FUNCTION_BLOCK L3_PlatoDivisor EXTENDS L1_ModuleBase

VAR_OUTPUT	
	fbController	: L2_PlatoDivisor_SFC:=(dr:=dr);  
	d0 				: L1_Sensor := (uiValue:= TRUE);
    D_1       		: L1_Actuator;
    E_1       		: L1_Actuator;
	NumGiros 		: DINT := 0;
	Angulo			: REAL := 0;
END_VAR

VAR
	AnguloAnim		: REAL := 0;
END_VAR

METHOD ProcessCycle : BOOL 

VAR_INPUT
	dr			: REFERENCE TO L1_Director;
	tapas		: REFERENCE TO L6_Tapas;	
END_VAR
IF dr.gmModeActual = L1_GEMMA.A6Inicializando THEN
	NumGiros := 0;
	Angulo	 := 0; // -45.0;
ELSE
	// Sensores y condiciones iniciales
	d0.ProcessCycle(LocalHost:=dr.gmLocalHost, sfcValue=>fbController.d0);
	IC := d0.uiValue;
	
	// Controlador
	fbController.ProcessCycle(dr.gmModeActual);
	fbController(
		dr:=dr, IC:=IC, Execute:=Execute, Ack:=Ack, Ready=>Ready, Done=>Done);
	IF fbController.Done AND NOT fbController.Performed THEN
		fbController.Performed 	:= TRUE;
		NumGiros 				:= NumGiros + 1;
		AnguloAnim				:= 0;		
	ELSIF fbController.Executing AND anguloanim >-35.0 THEN  
		AnguloAnim 	:= anguloanim - 0.2;	
	END_IF	
	Angulo 					:= AnguloAnim -45.0 * (NumGiros MOD 8); // 
	// Actuadores y actualización de tapas
	D_1.ProcessCycle(gmMode:=dr.gmModeActual, sfcValue:=fbController.D_1);
	E_1.ProcessCycle(gmMode:=dr.gmModeActual, sfcValue:=fbController.E_1);
END_IF
END_METHOD

END_FUNCTION_BLOCK

(* stored: Version 1.1.0.1, ProductVersion 3.1.4024.11
   POU L3_PlatoDivisor: Id {c71a4a01-3eb1-443b-a07e-accb57d2980d}, SpecialFunc None
   Method ProcessCycle: Id {a7156aed-454d-425e-80f1-664f90d71526} *)
